KUKA KRL data list: get_best_move.dat

&ACCESS RV1
DEFDAT  get_best_move PUBLIC

ENDDAT
